Staubli VAL3: place.pgx

program place(point pPosition, tool tTool, mdesc mApproach, mdesc mTarget)
  local point pOffset
begin

  // Función para soltar la pieza en el lugar deseado
  pOffset=appro(pPosition,{0,0,-50,0,0,0})
  // Se aproxima al destino
  movej(pOffset,tTool,mApproach)
  movel(pPosition,tTool,mTarget)
  open(tTool)
  movel(pOffset,tTool,mTarget)

end
